DECL LDAT LCPDATP325={VEL 1,ACC 100,APO_DIST 5,APO_FAC 50.0,ORI_TYP #VAR,CIRC_TYP #BASE,JERK_FAC 50.0}
DECL FDAT FP325={TOOL_NO 2,BASE_NO 10,IPO_FRAME #BASE,POINT2[] " ",TQ_STATE FALSE}
DECL E6POS XP325={X -66.960,Y 123.330,Z -48.800,A 0.000,B 0.000,C -0.000}
DECL LDAT LCPDATC326={VEL 0.1,ACC 100,APO_DIST 5,APO_FAC 50.0,ORI_TYP #VAR,CIRC_TYP #BASE,JERK_FAC 50.0}
DECL FDAT FC326={TOOL_NO 2,BASE_NO 10,IPO_FRAME #BASE,POINT2[] " ",TQ_STATE FALSE}
DECL E6POS XCAux326={X -53.710,Y 129.660,Z -48.800,A 0.000,B 0.000,C -0.000}
DECL E6POS XCDes326={X 53.710,Y 129.660,Z -48.800,A 0.000,B 0.000,C -0.000}
DECL LDAT LCPDATP327={VEL 1,ACC 100,APO_DIST 5,APO_FAC 50.0,ORI_TYP #VAR,CIRC_TYP #BASE,JERK_FAC 50.0}
DECL FDAT FP327={TOOL_NO 2,BASE_NO 10,IPO_FRAME #BASE,POINT2[] " ",TQ_STATE FALSE}
DECL E6POS XP327={X 66.960,Y 123.330,Z -48.800,A 0.000,B 0.000,C -0.000}
DECL LDAT LCPDATP328={VEL 1,ACC 100,APO_DIST 5,APO_FAC 50.0,ORI_TYP #VAR,CIRC_TYP #BASE,JERK_FAC 50.0}
DECL FDAT FP328={TOOL_NO 2,BASE_NO 10,IPO_FRAME #BASE,POINT2[] " ",TQ_STATE FALSE}
DECL E6POS XP328={X 67.920,Y 125.090,Z -48.800,A 0.000,B 0.000,C -0.000}
DECL LDAT LCPDATC329={VEL 0.1,ACC 100,APO_DIST 5,APO_FAC 50.0,ORI_TYP #VAR,CIRC_TYP #BASE,JERK_FAC 50.0}
DECL FDAT FC329={TOOL_NO 2,BASE_NO 10,IPO_FRAME #BASE,POINT2[] " ",TQ_STATE FALSE}
DECL E6POS XCAux329={X 54.470,Y 131.500,Z -48.800,A 0.000,B 0.000,C -0.000}
DECL E6POS XCDes329={X -54.470,Y 131.500,Z -48.800,A 0.000,B 0.000,C -0.000}
DECL LDAT LCPDATP330={VEL 1,ACC 100,APO_DIST 5,APO_FAC 50.0,ORI_TYP #VAR,CIRC_TYP #BASE,JERK_FAC 50.0}
DECL FDAT FP330={TOOL_NO 2,BASE_NO 10,IPO_FRAME #BASE,POINT2[] " ",TQ_STATE FALSE}
DECL E6POS XP330={X -67.920,Y 125.090,Z -48.800,A 0.000,B 0.000,C -0.000}
DECL LDAT LCPDATP331={VEL 1,ACC 100,APO_DIST 5,APO_FAC 50.0,ORI_TYP #VAR,CIRC_TYP #BASE,JERK_FAC 50.0}
DECL FDAT FP331={TOOL_NO 2,BASE_NO 10,IPO_FRAME #BASE,POINT2[] " ",TQ_STATE FALSE}
DECL E6POS XP331={X -68.870,Y 126.850,Z -48.800,A 0.000,B 0.000,C -0.000}
DECL LDAT LCPDATC332={VEL 0.1,ACC 100,APO_DIST 5,APO_FAC 50.0,ORI_TYP #VAR,CIRC_TYP #BASE,JERK_FAC 50.0}
DECL FDAT FC332={TOOL_NO 2,BASE_NO 10,IPO_FRAME #BASE,POINT2[] " ",TQ_STATE FALSE}
DECL E6POS XCAux332={X -55.240,Y 133.350,Z -48.800,A 0.000,B 0.000,C -0.000}
DECL E6POS XCDes332={X 55.240,Y 133.350,Z -48.800,A 0.000,B 0.000,C -0.000}
DECL LDAT LCPDATP333={VEL 1,ACC 100,APO_DIST 5,APO_FAC 50.0,ORI_TYP #VAR,CIRC_TYP #BASE,JERK_FAC 50.0}
DECL FDAT FP333={TOOL_NO 2,BASE_NO 10,IPO_FRAME #BASE,POINT2[] " ",TQ_STATE FALSE}
DECL E6POS XP333={X 68.870,Y 126.850,Z -48.800,A 0.000,B 0.000,C -0.000}
DECL LDAT LCPDATP334={VEL 1,ACC 100,APO_DIST 5,APO_FAC 50.0,ORI_TYP #VAR,CIRC_TYP #BASE,JERK_FAC 50.0}
DECL FDAT FP334={TOOL_NO 2,BASE_NO 10,IPO_FRAME #BASE,POINT2[] " ",TQ_STATE FALSE}
DECL E6POS XP334={X 69.830,Y 128.610,Z -48.800,A 0.000,B 0.000,C -0.000}
DECL LDAT LCPDATC335={VEL 0.1,ACC 100,APO_DIST 5,APO_FAC 50.0,ORI_TYP #VAR,CIRC_TYP #BASE,JERK_FAC 50.0}
DECL FDAT FC335={TOOL_NO 2,BASE_NO 10,IPO_FRAME #BASE,POINT2[] " ",TQ_STATE FALSE}
DECL E6POS XCAux335={X 56.000,Y 135.200,Z -48.800,A 0.000,B 0.000,C -0.000}
DECL E6POS XCDes335={X -56.000,Y 135.200,Z -48.800,A 0.000,B 0.000,C -0.000}
DECL LDAT LCPDATP336={VEL 1,ACC 100,APO_DIST 5,APO_FAC 50.0,ORI_TYP #VAR,CIRC_TYP #BASE,JERK_FAC 50.0}
DECL FDAT FP336={TOOL_NO 2,BASE_NO 10,IPO_FRAME #BASE,POINT2[] " ",TQ_STATE FALSE}
DECL E6POS XP336={X -69.830,Y 128.610,Z -48.800,A 0.000,B 0.000,C -0.000}
DECL LDAT LCPDATP337={VEL 1,ACC 100,APO_DIST 5,APO_FAC 50.0,ORI_TYP #VAR,CIRC_TYP #BASE,JERK_FAC 50.0}
DECL FDAT FP337={TOOL_NO 2,BASE_NO 10,IPO_FRAME #BASE,POINT2[] " ",TQ_STATE FALSE}
DECL E6POS XP337={X -70.780,Y 130.360,Z -48.800,A 0.000,B 0.000,C -0.000}
DECL LDAT LCPDATC338={VEL 0.1,ACC 100,APO_DIST 5,APO_FAC 50.0,ORI_TYP #VAR,CIRC_TYP #BASE,JERK_FAC 50.0}
DECL FDAT FC338={TOOL_NO 2,BASE_NO 10,IPO_FRAME #BASE,POINT2[] " ",TQ_STATE FALSE}
DECL E6POS XCAux338={X -56.770,Y 137.050,Z -48.800,A 0.000,B 0.000,C -0.000}
DECL E6POS XCDes338={X 56.770,Y 137.050,Z -48.800,A 0.000,B 0.000,C -0.000}
DECL LDAT LCPDATP339={VEL 1,ACC 100,APO_DIST 5,APO_FAC 50.0,ORI_TYP #VAR,CIRC_TYP #BASE,JERK_FAC 50.0}
DECL FDAT FP339={TOOL_NO 2,BASE_NO 10,IPO_FRAME #BASE,POINT2[] " ",TQ_STATE FALSE}
DECL E6POS XP339={X 70.780,Y 130.360,Z -48.800,A 0.000,B 0.000,C -0.000}
DECL LDAT LCPDATP340={VEL 1,ACC 100,APO_DIST 5,APO_FAC 50.0,ORI_TYP #VAR,CIRC_TYP #BASE,JERK_FAC 50.0}
DECL FDAT FP340={TOOL_NO 2,BASE_NO 10,IPO_FRAME #BASE,POINT2[] " ",TQ_STATE FALSE}
DECL E6POS XP340={X 71.740,Y 132.120,Z -48.800,A 0.000,B 0.000,C -0.000}
DECL LDAT LCPDATC341={VEL 0.1,ACC 100,APO_DIST 5,APO_FAC 50.0,ORI_TYP #VAR,CIRC_TYP #BASE,JERK_FAC 50.0}
DECL FDAT FC341={TOOL_NO 2,BASE_NO 10,IPO_FRAME #BASE,POINT2[] " ",TQ_STATE FALSE}
DECL E6POS XCAux341={X 57.530,Y 138.890,Z -48.800,A 0.000,B 0.000,C -0.000}
DECL E6POS XCDes341={X -57.530,Y 138.890,Z -48.800,A 0.000,B 0.000,C -0.000}
DECL LDAT LCPDATP342={VEL 1,ACC 100,APO_DIST 5,APO_FAC 50.0,ORI_TYP #VAR,CIRC_TYP #BASE,JERK_FAC 50.0}
DECL FDAT FP342={TOOL_NO 2,BASE_NO 10,IPO_FRAME #BASE,POINT2[] " ",TQ_STATE FALSE}
DECL E6POS XP342={X -71.740,Y 132.120,Z -48.800,A 0.000,B 0.000,C -0.000}
DECL LDAT LCPDATP343={VEL 1,ACC 100,APO_DIST 5,APO_FAC 50.0,ORI_TYP #VAR,CIRC_TYP #BASE,JERK_FAC 50.0}
DECL FDAT FP343={TOOL_NO 2,BASE_NO 10,IPO_FRAME #BASE,POINT2[] " ",TQ_STATE FALSE}
DECL E6POS XP343={X -69.340,Y 127.710,Z -48.400,A 0.000,B -3.840,C -7.100}
DECL LDAT LCPDATC344={VEL 0.1,ACC 100,APO_DIST 5,APO_FAC 50.0,ORI_TYP #VAR,CIRC_TYP #BASE,JERK_FAC 50.0}
DECL FDAT FC344={TOOL_NO 2,BASE_NO 10,IPO_FRAME #BASE,POINT2[] " ",TQ_STATE FALSE}
DECL E6POS XCAux344={X -55.610,Y 134.260,Z -48.400,A 0.000,B -3.080,C -7.460}
DECL E6POS XCDes344={X 55.610,Y 134.260,Z -48.400,A 0.000,B 3.080,C -7.460}
DECL LDAT LCPDATP345={VEL 1,ACC 100,APO_DIST 5,APO_FAC 50.0,ORI_TYP #VAR,CIRC_TYP #BASE,JERK_FAC 50.0}
DECL FDAT FP345={TOOL_NO 2,BASE_NO 10,IPO_FRAME #BASE,POINT2[] " ",TQ_STATE FALSE}
DECL E6POS XP345={X 69.340,Y 127.710,Z -48.400,A 0.000,B 3.840,C -7.100}
DECL LDAT LCPDATP346={VEL 1,ACC 100,APO_DIST 5,APO_FAC 50.0,ORI_TYP #VAR,CIRC_TYP #BASE,JERK_FAC 50.0}
DECL FDAT FP346={TOOL_NO 2,BASE_NO 10,IPO_FRAME #BASE,POINT2[] " ",TQ_STATE FALSE}
DECL E6POS XP346={X 65.420,Y 120.500,Z -46.340,A -0.000,B 9.430,C -17.800}
DECL LDAT LCPDATC347={VEL 0.1,ACC 100,APO_DIST 5,APO_FAC 50.0,ORI_TYP #VAR,CIRC_TYP #BASE,JERK_FAC 50.0}
DECL FDAT FC347={TOOL_NO 2,BASE_NO 10,IPO_FRAME #BASE,POINT2[] " ",TQ_STATE FALSE}
DECL E6POS XCAux347={X 52.470,Y 126.680,Z -46.340,A -0.000,B 7.550,C -18.660}
DECL E6POS XCDes347={X -52.470,Y 126.680,Z -46.340,A -0.000,B -7.550,C -18.660}
DECL LDAT LCPDATP348={VEL 1,ACC 100,APO_DIST 5,APO_FAC 50.0,ORI_TYP #VAR,CIRC_TYP #BASE,JERK_FAC 50.0}
DECL FDAT FP348={TOOL_NO 2,BASE_NO 10,IPO_FRAME #BASE,POINT2[] " ",TQ_STATE FALSE}
DECL E6POS XP348={X -65.420,Y 120.500,Z -46.340,A -0.000,B -9.430,C -17.800}
DECL LDAT LCPDATP349={VEL 1,ACC 100,APO_DIST 5,APO_FAC 50.0,ORI_TYP #VAR,CIRC_TYP #BASE,JERK_FAC 50.0}
DECL FDAT FP349={TOOL_NO 2,BASE_NO 10,IPO_FRAME #BASE,POINT2[] " ",TQ_STATE FALSE}
DECL E6POS XP349={X -61.800,Y 113.820,Z -42.620,A -0.000,B -14.680,C -28.850}
DECL LDAT LCPDATC350={VEL 0.1,ACC 100,APO_DIST 5,APO_FAC 50.0,ORI_TYP #VAR,CIRC_TYP #BASE,JERK_FAC 50.0}
DECL FDAT FC350={TOOL_NO 2,BASE_NO 10,IPO_FRAME #BASE,POINT2[] " ",TQ_STATE FALSE}
DECL E6POS XCAux350={X -49.560,Y 119.650,Z -42.620,A 0.000,B -11.730,C -30.080}
DECL E6POS XCDes350={X 49.560,Y 119.650,Z -42.620,A -0.000,B 11.730,C -30.080}
DECL LDAT LCPDATP351={VEL 1,ACC 100,APO_DIST 5,APO_FAC 50.0,ORI_TYP #VAR,CIRC_TYP #BASE,JERK_FAC 50.0}
DECL FDAT FP351={TOOL_NO 2,BASE_NO 10,IPO_FRAME #BASE,POINT2[] " ",TQ_STATE FALSE}
DECL E6POS XP351={X 61.800,Y 113.820,Z -42.620,A 0.000,B 14.680,C -28.850}
DECL LDAT LCPDATP352={VEL 1,ACC 100,APO_DIST 5,APO_FAC 50.0,ORI_TYP #VAR,CIRC_TYP #BASE,JERK_FAC 50.0}
DECL FDAT FP352={TOOL_NO 2,BASE_NO 10,IPO_FRAME #BASE,POINT2[] " ",TQ_STATE FALSE}
DECL E6POS XP352={X 58.620,Y 107.960,Z -37.400,A 0.000,B 19.390,C -40.410}
DECL LDAT LCPDATC353={VEL 0.1,ACC 100,APO_DIST 5,APO_FAC 50.0,ORI_TYP #VAR,CIRC_TYP #BASE,JERK_FAC 50.0}
DECL FDAT FC353={TOOL_NO 2,BASE_NO 10,IPO_FRAME #BASE,POINT2[] " ",TQ_STATE FALSE}
DECL E6POS XCAux353={X 47.010,Y 113.500,Z -37.400,A -0.000,B 15.440,C -41.830}
DECL E6POS XCDes353={X -47.010,Y 113.500,Z -37.400,A -0.000,B -15.440,C -41.830}
DECL LDAT LCPDATP354={VEL 1,ACC 100,APO_DIST 5,APO_FAC 50.0,ORI_TYP #VAR,CIRC_TYP #BASE,JERK_FAC 50.0}
DECL FDAT FP354={TOOL_NO 2,BASE_NO 10,IPO_FRAME #BASE,POINT2[] " ",TQ_STATE FALSE}
DECL E6POS XP354={X -58.620,Y 107.960,Z -37.400,A 0.000,B -19.390,C -40.410}
DECL LDAT LCPDATP355={VEL 1,ACC 100,APO_DIST 5,APO_FAC 50.0,ORI_TYP #VAR,CIRC_TYP #BASE,JERK_FAC 50.0}
DECL FDAT FP355={TOOL_NO 2,BASE_NO 10,IPO_FRAME #BASE,POINT2[] " ",TQ_STATE FALSE}
DECL E6POS XP355={X -59.520,Y 109.620,Z -39.640,A 0.000,B -17.860,C -36.410}
DECL LDAT LCPDATC356={VEL 0.1,ACC 100,APO_DIST 5,APO_FAC 50.0,ORI_TYP #VAR,CIRC_TYP #BASE,JERK_FAC 50.0}
DECL FDAT FC356={TOOL_NO 2,BASE_NO 10,IPO_FRAME #BASE,POINT2[] " ",TQ_STATE FALSE}
DECL E6POS XCAux356={X -47.730,Y 115.240,Z -39.640,A 0.000,B -14.240,C -37.780}
DECL E6POS XCDes356={X 47.730,Y 115.240,Z -39.640,A 0.000,B 14.240,C -37.780}
DECL LDAT LCPDATP357={VEL 1,ACC 100,APO_DIST 5,APO_FAC 50.0,ORI_TYP #VAR,CIRC_TYP #BASE,JERK_FAC 50.0}
DECL FDAT FP357={TOOL_NO 2,BASE_NO 10,IPO_FRAME #BASE,POINT2[] " ",TQ_STATE FALSE}
DECL E6POS XP357={X 59.520,Y 109.620,Z -39.640,A 0.000,B 17.860,C -36.410}
DECL LDAT LCPDATP358={VEL 1,ACC 100,APO_DIST 5,APO_FAC 50.0,ORI_TYP #VAR,CIRC_TYP #BASE,JERK_FAC 50.0}
DECL FDAT FP358={TOOL_NO 2,BASE_NO 10,IPO_FRAME #BASE,POINT2[] " ",TQ_STATE FALSE}
DECL E6POS XP358={X 63.060,Y 116.140,Z -44.590,A 0.000,B 12.710,C -24.550}
DECL LDAT LCPDATC359={VEL 0.1,ACC 100,APO_DIST 5,APO_FAC 50.0,ORI_TYP #VAR,CIRC_TYP #BASE,JERK_FAC 50.0}
DECL FDAT FC359={TOOL_NO 2,BASE_NO 10,IPO_FRAME #BASE,POINT2[] " ",TQ_STATE FALSE}
DECL E6POS XCAux359={X 50.570,Y 122.100,Z -44.590,A 0.000,B 10.170,C -25.650}
DECL E6POS XCDes359={X -50.570,Y 122.100,Z -44.590,A 0.000,B -10.170,C -25.650}
DECL LDAT LCPDATP360={VEL 1,ACC 100,APO_DIST 5,APO_FAC 50.0,ORI_TYP #VAR,CIRC_TYP #BASE,JERK_FAC 50.0}
DECL FDAT FP360={TOOL_NO 2,BASE_NO 10,IPO_FRAME #BASE,POINT2[] " ",TQ_STATE FALSE}
DECL E6POS XP360={X -63.060,Y 116.140,Z -44.590,A -0.000,B -12.710,C -24.550}
DECL LDAT LCPDATP361={VEL 1,ACC 100,APO_DIST 5,APO_FAC 50.0,ORI_TYP #VAR,CIRC_TYP #BASE,JERK_FAC 50.0}
DECL FDAT FP361={TOOL_NO 2,BASE_NO 10,IPO_FRAME #BASE,POINT2[] " ",TQ_STATE FALSE}
DECL E6POS XP361={X -67.030,Y 123.450,Z -47.820,A -0.000,B -7.060,C -13.190}
DECL LDAT LCPDATC362={VEL 0.1,ACC 100,APO_DIST 5,APO_FAC 50.0,ORI_TYP #VAR,CIRC_TYP #BASE,JERK_FAC 50.0}
DECL FDAT FC362={TOOL_NO 2,BASE_NO 10,IPO_FRAME #BASE,POINT2[] " ",TQ_STATE FALSE}
DECL E6POS XCAux362={X -53.760,Y 129.780,Z -47.820,A 0.000,B -5.660,C -13.840}
DECL E6POS XCDes362={X 53.760,Y 129.780,Z -47.820,A 0.000,B 5.660,C -13.840}
DECL LDAT LCPDATP363={VEL 1,ACC 100,APO_DIST 5,APO_FAC 50.0,ORI_TYP #VAR,CIRC_TYP #BASE,JERK_FAC 50.0}
DECL FDAT FP363={TOOL_NO 2,BASE_NO 10,IPO_FRAME #BASE,POINT2[] " ",TQ_STATE FALSE}
DECL E6POS XP363={X 67.030,Y 123.450,Z -47.820,A 0.000,B 7.060,C -13.190}
DECL LDAT LCPDATP364={VEL 1,ACC 100,APO_DIST 5,APO_FAC 50.0,ORI_TYP #VAR,CIRC_TYP #BASE,JERK_FAC 50.0}
DECL FDAT FP364={TOOL_NO 2,BASE_NO 10,IPO_FRAME #BASE,POINT2[] " ",TQ_STATE FALSE}
DECL E6POS XP364={X 71.240,Y 131.200,Z -49.160,A 0.000,B 1.140,C -2.110}
DECL LDAT LCPDATC365={VEL 0.1,ACC 100,APO_DIST 5,APO_FAC 50.0,ORI_TYP #VAR,CIRC_TYP #BASE,JERK_FAC 50.0}
DECL FDAT FC365={TOOL_NO 2,BASE_NO 10,IPO_FRAME #BASE,POINT2[] " ",TQ_STATE FALSE}
DECL E6POS XCAux365={X 57.130,Y 137.930,Z -49.160,A 0.000,B 0.920,C -2.210}
DECL E6POS XCDes365={X -57.130,Y 137.930,Z -49.160,A 0.000,B -0.920,C -2.210}
DECL LDAT LCPDATP366={VEL 1,ACC 100,APO_DIST 5,APO_FAC 50.0,ORI_TYP #VAR,CIRC_TYP #BASE,JERK_FAC 50.0}
DECL FDAT FP366={TOOL_NO 2,BASE_NO 10,IPO_FRAME #BASE,POINT2[] " ",TQ_STATE FALSE}
DECL E6POS XP366={X -71.240,Y 131.200,Z -49.160,A 0.000,B -1.140,C -2.110}
DECL LDAT LCPDATP367={VEL 1,ACC 100,APO_DIST 5,APO_FAC 50.0,ORI_TYP #VAR,CIRC_TYP #BASE,JERK_FAC 50.0}
DECL FDAT FP367={TOOL_NO 2,BASE_NO 10,IPO_FRAME #BASE,POINT2[] " ",TQ_STATE FALSE}
DECL E6POS XP367={X -71.280,Y 131.280,Z -49.200,A 0.000,B 0.000,C -0.000}
DECL LDAT LCPDATC368={VEL 0.1,ACC 100,APO_DIST 5,APO_FAC 50.0,ORI_TYP #VAR,CIRC_TYP #BASE,JERK_FAC 50.0}
DECL FDAT FC368={TOOL_NO 2,BASE_NO 10,IPO_FRAME #BASE,POINT2[] " ",TQ_STATE FALSE}
DECL E6POS XCAux368={X -57.170,Y 138.010,Z -49.200,A 0.000,B 0.000,C -0.000}
DECL E6POS XCDes368={X 57.170,Y 138.010,Z -49.200,A 0.000,B 0.000,C -0.000}
DECL LDAT LCPDATP369={VEL 1,ACC 100,APO_DIST 5,APO_FAC 50.0,ORI_TYP #VAR,CIRC_TYP #BASE,JERK_FAC 50.0}
DECL FDAT FP369={TOOL_NO 2,BASE_NO 10,IPO_FRAME #BASE,POINT2[] " ",TQ_STATE FALSE}
DECL E6POS XP369={X 71.280,Y 131.280,Z -49.200,A 0.000,B 0.000,C -0.000}
DECL LDAT LCPDATP370={VEL 1,ACC 100,APO_DIST 5,APO_FAC 50.0,ORI_TYP #VAR,CIRC_TYP #BASE,JERK_FAC 50.0}
DECL FDAT FP370={TOOL_NO 2,BASE_NO 10,IPO_FRAME #BASE,POINT2[] " ",TQ_STATE FALSE}
DECL E6POS XP370={X 70.320,Y 129.520,Z -49.200,A 0.000,B 0.000,C -0.000}
DECL LDAT LCPDATC371={VEL 0.1,ACC 100,APO_DIST 5,APO_FAC 50.0,ORI_TYP #VAR,CIRC_TYP #BASE,JERK_FAC 50.0}
DECL FDAT FC371={TOOL_NO 2,BASE_NO 10,IPO_FRAME #BASE,POINT2[] " ",TQ_STATE FALSE}
DECL E6POS XCAux371={X 56.400,Y 136.160,Z -49.200,A 0.000,B 0.000,C -0.000}
DECL E6POS XCDes371={X -56.400,Y 136.160,Z -49.200,A 0.000,B 0.000,C -0.000}
DECL LDAT LCPDATP372={VEL 1,ACC 100,APO_DIST 5,APO_FAC 50.0,ORI_TYP #VAR,CIRC_TYP #BASE,JERK_FAC 50.0}
DECL FDAT FP372={TOOL_NO 2,BASE_NO 10,IPO_FRAME #BASE,POINT2[] " ",TQ_STATE FALSE}
DECL E6POS XP372={X -70.320,Y 129.520,Z -49.200,A 0.000,B 0.000,C -0.000}
DECL LDAT LCPDATP373={VEL 1,ACC 100,APO_DIST 5,APO_FAC 50.0,ORI_TYP #VAR,CIRC_TYP #BASE,JERK_FAC 50.0}
DECL FDAT FP373={TOOL_NO 2,BASE_NO 10,IPO_FRAME #BASE,POINT2[] " ",TQ_STATE FALSE}
DECL E6POS XP373={X -69.370,Y 127.760,Z -49.200,A 0.000,B 0.000,C -0.000}
DECL LDAT LCPDATC374={VEL 0.1,ACC 100,APO_DIST 5,APO_FAC 50.0,ORI_TYP #VAR,CIRC_TYP #BASE,JERK_FAC 50.0}
DECL FDAT FC374={TOOL_NO 2,BASE_NO 10,IPO_FRAME #BASE,POINT2[] " ",TQ_STATE FALSE}
DECL E6POS XCAux374={X -55.640,Y 134.320,Z -49.200,A 0.000,B 0.000,C -0.000}
DECL E6POS XCDes374={X 55.640,Y 134.320,Z -49.200,A 0.000,B 0.000,C -0.000}
DECL LDAT LCPDATP375={VEL 1,ACC 100,APO_DIST 5,APO_FAC 50.0,ORI_TYP #VAR,CIRC_TYP #BASE,JERK_FAC 50.0}
DECL FDAT FP375={TOOL_NO 2,BASE_NO 10,IPO_FRAME #BASE,POINT2[] " ",TQ_STATE FALSE}
DECL E6POS XP375={X 69.370,Y 127.760,Z -49.200,A 0.000,B 0.000,C -0.000}
DECL LDAT LCPDATP376={VEL 1,ACC 100,APO_DIST 5,APO_FAC 50.0,ORI_TYP #VAR,CIRC_TYP #BASE,JERK_FAC 50.0}
DECL FDAT FP376={TOOL_NO 2,BASE_NO 10,IPO_FRAME #BASE,POINT2[] " ",TQ_STATE FALSE}
DECL E6POS XP376={X 68.420,Y 126.010,Z -49.200,A 0.000,B 0.000,C -0.000}
DECL LDAT LCPDATC377={VEL 0.1,ACC 100,APO_DIST 5,APO_FAC 50.0,ORI_TYP #VAR,CIRC_TYP #BASE,JERK_FAC 50.0}
DECL FDAT FC377={TOOL_NO 2,BASE_NO 10,IPO_FRAME #BASE,POINT2[] " ",TQ_STATE FALSE}
DECL E6POS XCAux377={X 54.870,Y 132.470,Z -49.200,A 0.000,B 0.000,C -0.000}
DECL E6POS XCDes377={X -54.870,Y 132.470,Z -49.200,A 0.000,B 0.000,C -0.000}
DECL LDAT LCPDATP378={VEL 1,ACC 100,APO_DIST 5,APO_FAC 50.0,ORI_TYP #VAR,CIRC_TYP #BASE,JERK_FAC 50.0}
DECL FDAT FP378={TOOL_NO 2,BASE_NO 10,IPO_FRAME #BASE,POINT2[] " ",TQ_STATE FALSE}
DECL E6POS XP378={X -68.420,Y 126.010,Z -49.200,A 0.000,B 0.000,C -0.000}
DECL LDAT LCPDATP379={VEL 1,ACC 100,APO_DIST 5,APO_FAC 50.0,ORI_TYP #VAR,CIRC_TYP #BASE,JERK_FAC 50.0}
DECL FDAT FP379={TOOL_NO 2,BASE_NO 10,IPO_FRAME #BASE,POINT2[] " ",TQ_STATE FALSE}
DECL E6POS XP379={X -67.460,Y 124.250,Z -49.200,A 0.000,B 0.000,C -0.000}
DECL LDAT LCPDATC380={VEL 0.1,ACC 100,APO_DIST 5,APO_FAC 50.0,ORI_TYP #VAR,CIRC_TYP #BASE,JERK_FAC 50.0}
DECL FDAT FC380={TOOL_NO 2,BASE_NO 10,IPO_FRAME #BASE,POINT2[] " ",TQ_STATE FALSE}
DECL E6POS XCAux380={X -54.100,Y 130.620,Z -49.200,A 0.000,B 0.000,C -0.000}
DECL E6POS XCDes380={X 54.100,Y 130.620,Z -49.200,A 0.000,B 0.000,C -0.000}
DECL LDAT LCPDATP381={VEL 1,ACC 100,APO_DIST 5,APO_FAC 50.0,ORI_TYP #VAR,CIRC_TYP #BASE,JERK_FAC 50.0}
DECL FDAT FP381={TOOL_NO 2,BASE_NO 10,IPO_FRAME #BASE,POINT2[] " ",TQ_STATE FALSE}
DECL E6POS XP381={X 67.460,Y 124.250,Z -49.200,A 0.000,B 0.000,C -0.000}
DECL LDAT LCPDATP382={VEL 1,ACC 100,APO_DIST 5,APO_FAC 50.0,ORI_TYP #VAR,CIRC_TYP #BASE,JERK_FAC 50.0}
DECL FDAT FP382={TOOL_NO 2,BASE_NO 10,IPO_FRAME #BASE,POINT2[] " ",TQ_STATE FALSE}
DECL E6POS XP382={X 66.510,Y 122.490,Z -49.200,A 0.000,B 0.000,C -0.000}
DECL LDAT LCPDATC383={VEL 0.1,ACC 100,APO_DIST 5,APO_FAC 50.0,ORI_TYP #VAR,CIRC_TYP #BASE,JERK_FAC 50.0}
DECL FDAT FC383={TOOL_NO 2,BASE_NO 10,IPO_FRAME #BASE,POINT2[] " ",TQ_STATE FALSE}
DECL E6POS XCAux383={X 53.340,Y 128.770,Z -49.200,A 0.000,B 0.000,C -0.000}
DECL E6POS XCDes383={X -53.340,Y 128.770,Z -49.200,A 0.000,B 0.000,C -0.000}
DECL LDAT LCPDATP384={VEL 1,ACC 100,APO_DIST 5,APO_FAC 50.0,ORI_TYP #VAR,CIRC_TYP #BASE,JERK_FAC 50.0}
DECL FDAT FP384={TOOL_NO 2,BASE_NO 10,IPO_FRAME #BASE,POINT2[] " ",TQ_STATE FALSE}
DECL E6POS XP384={X -66.510,Y 122.490,Z -49.200,A 0.000,B 0.000,C -0.000}
DECL LDAT LCPDATP385={VEL 1,ACC 100,APO_DIST 5,APO_FAC 50.0,ORI_TYP #VAR,CIRC_TYP #BASE,JERK_FAC 50.0}
DECL FDAT FP385={TOOL_NO 2,BASE_NO 10,IPO_FRAME #BASE,POINT2[] " ",TQ_STATE FALSE}
DECL E6POS XP385={X -69.770,Y 128.510,Z -48.560,A -0.000,B 4.840,C 8.980}
DECL LDAT LCPDATC386={VEL 0.1,ACC 100,APO_DIST 5,APO_FAC 50.0,ORI_TYP #VAR,CIRC_TYP #BASE,JERK_FAC 50.0}
DECL FDAT FC386={TOOL_NO 2,BASE_NO 10,IPO_FRAME #BASE,POINT2[] " ",TQ_STATE FALSE}
DECL E6POS XCAux386={X -55.960,Y 135.100,Z -48.560,A -0.000,B 3.880,C 9.430}
DECL E6POS XCDes386={X 55.960,Y 135.100,Z -48.560,A 0.000,B -3.880,C 9.430}
DECL LDAT LCPDATP387={VEL 1,ACC 100,APO_DIST 5,APO_FAC 50.0,ORI_TYP #VAR,CIRC_TYP #BASE,JERK_FAC 50.0}
DECL FDAT FP387={TOOL_NO 2,BASE_NO 10,IPO_FRAME #BASE,POINT2[] " ",TQ_STATE FALSE}
DECL E6POS XP387={X 69.770,Y 128.510,Z -48.560,A 0.000,B -4.840,C 8.980}
DECL LDAT LCPDATP388={VEL 1,ACC 100,APO_DIST 5,APO_FAC 50.0,ORI_TYP #VAR,CIRC_TYP #BASE,JERK_FAC 50.0}
DECL FDAT FP388={TOOL_NO 2,BASE_NO 10,IPO_FRAME #BASE,POINT2[] " ",TQ_STATE FALSE}
DECL E6POS XP388={X 73.860,Y 136.030,Z -46.030,A 0.000,B -10.620,C 20.210}
DECL LDAT LCPDATC389={VEL 0.1,ACC 100,APO_DIST 5,APO_FAC 50.0,ORI_TYP #VAR,CIRC_TYP #BASE,JERK_FAC 50.0}
DECL FDAT FC389={TOOL_NO 2,BASE_NO 10,IPO_FRAME #BASE,POINT2[] " ",TQ_STATE FALSE}
DECL E6POS XCAux389={X 59.230,Y 143.000,Z -46.030,A -0.000,B -8.500,C 21.150}
DECL E6POS XCDes389={X -59.230,Y 143.000,Z -46.030,A 0.000,B 8.500,C 21.150}
DECL LDAT LCPDATP390={VEL 1,ACC 100,APO_DIST 5,APO_FAC 50.0,ORI_TYP #VAR,CIRC_TYP #BASE,JERK_FAC 50.0}
DECL FDAT FP390={TOOL_NO 2,BASE_NO 10,IPO_FRAME #BASE,POINT2[] " ",TQ_STATE FALSE}
DECL E6POS XP390={X -73.860,Y 136.030,Z -46.030,A -0.000,B 10.620,C 20.210}
DECL LDAT LCPDATP391={VEL 1,ACC 100,APO_DIST 5,APO_FAC 50.0,ORI_TYP #VAR,CIRC_TYP #BASE,JERK_FAC 50.0}
DECL FDAT FP391={TOOL_NO 2,BASE_NO 10,IPO_FRAME #BASE,POINT2[] " ",TQ_STATE FALSE}
DECL E6POS XP391={X -77.580,Y 142.880,Z -41.700,A 0.000,B 15.990,C 31.850}
DECL LDAT LCPDATC392={VEL 0.1,ACC 100,APO_DIST 5,APO_FAC 50.0,ORI_TYP #VAR,CIRC_TYP #BASE,JERK_FAC 50.0}
DECL FDAT FC392={TOOL_NO 2,BASE_NO 10,IPO_FRAME #BASE,POINT2[] " ",TQ_STATE FALSE}
DECL E6POS XCAux392={X -62.220,Y 150.210,Z -41.700,A 0.000,B 12.760,C 33.150}
DECL E6POS XCDes392={X 62.220,Y 150.210,Z -41.700,A 0.000,B -12.760,C 33.150}
DECL LDAT LCPDATP393={VEL 1,ACC 100,APO_DIST 5,APO_FAC 50.0,ORI_TYP #VAR,CIRC_TYP #BASE,JERK_FAC 50.0}
DECL FDAT FP393={TOOL_NO 2,BASE_NO 10,IPO_FRAME #BASE,POINT2[] " ",TQ_STATE FALSE}
DECL E6POS XP393={X 77.580,Y 142.880,Z -41.700,A 0.000,B -15.990,C 31.850}
DECL LDAT LCPDATP394={VEL 1,ACC 100,APO_DIST 5,APO_FAC 50.0,ORI_TYP #VAR,CIRC_TYP #BASE,JERK_FAC 50.0}
DECL FDAT FP394={TOOL_NO 2,BASE_NO 10,IPO_FRAME #BASE,POINT2[] " ",TQ_STATE FALSE}
DECL E6POS XP394={X 80.770,Y 148.750,Z -35.790,A 0.000,B -20.700,C 44.100}
DECL LDAT LCPDATC395={VEL 0.1,ACC 100,APO_DIST 5,APO_FAC 50.0,ORI_TYP #VAR,CIRC_TYP #BASE,JERK_FAC 50.0}
DECL FDAT FC395={TOOL_NO 2,BASE_NO 10,IPO_FRAME #BASE,POINT2[] " ",TQ_STATE FALSE}
DECL E6POS XCAux395={X 64.770,Y 156.380,Z -35.790,A 0.000,B -16.470,C 45.530}
DECL E6POS XCDes395={X -64.770,Y 156.380,Z -35.790,A 0.000,B 16.470,C 45.530}
DECL LDAT LCPDATP396={VEL 1,ACC 100,APO_DIST 5,APO_FAC 50.0,ORI_TYP #VAR,CIRC_TYP #BASE,JERK_FAC 50.0}
DECL FDAT FP396={TOOL_NO 2,BASE_NO 10,IPO_FRAME #BASE,POINT2[] " ",TQ_STATE FALSE}
DECL E6POS XP396={X -80.770,Y 148.750,Z -35.790,A 0.000,B 20.700,C 44.100}
DECL LDAT LCPDATP397={VEL 0.5,ACC 100,APO_DIST 5,APO_FAC 50.0,ORI_TYP #VAR,CIRC_TYP #BASE,JERK_FAC 50.0}
DECL FDAT FP397={TOOL_NO 2,BASE_NO 10,IPO_FRAME #BASE,POINT2[] " ",TQ_STATE FALSE}
DECL E6POS XP397={X -113.090,Y 116.200,Z 97.800,A 0.000,B 0.000,C 180.000}
DECL LDAT LCPDATP398={VEL 0.5,ACC 100,APO_DIST 5,APO_FAC 50.0,ORI_TYP #VAR,CIRC_TYP #BASE,JERK_FAC 50.0}
DECL FDAT FP398={TOOL_NO 2,BASE_NO 10,IPO_FRAME #BASE,POINT2[] " ",TQ_STATE FALSE}
DECL E6POS XP398={X -113.090,Y 216.200,Z 97.800,A 0.000,B 0.000,C 180.000}
DECL LDAT LCPDATP399={VEL 1.0,ACC 100,APO_DIST 5,APO_FAC 50.0,ORI_TYP #VAR,CIRC_TYP #BASE,JERK_FAC 50.0}
DECL FDAT FP399={TOOL_NO 2,BASE_NO 10,IPO_FRAME #BASE,POINT2[] " ",TQ_STATE FALSE}
DECL E6POS XP399={X -113.090,Y 380.000,Z -20.000,A 0.000,B 0.000,C 0.000}
DECL LDAT LCPDATP400={VEL 1.0,ACC 100,APO_DIST 5,APO_FAC 50.0,ORI_TYP #VAR,CIRC_TYP #BASE,JERK_FAC 50.0}
DECL FDAT FP400={TOOL_NO 2,BASE_NO 10,IPO_FRAME #BASE,POINT2[] " ",TQ_STATE FALSE}
DECL E6POS XP400={X -60.500,Y 380.000,Z -20.000,A 0.000,B 0.000,C 0.000}
;ENDDAT for Routine_0

ENDDAT
